TYPE ST_EL70xx_STM_Control :
STRUCT
	Enable			AT %Q* : BIT;
	Reset			AT %Q* : BIT;
	ReduceTorque 	AT %Q* : BIT;	//Spulenstrom reduzieren
END_STRUCT
END_TYPE

(* stored: Version 1.1.0.1, ProductVersion 3.1.4024.11
   DUT ST_EL70xx_STM_Control: Id {f36d8772-2aca-478a-a5c3-5de42e561ac0} *)
